(* CoDeSys 2.3.9.62 project: Practica1Ej2.pro *)
(* Libraries: Standard.lib 4.10.05 11:14:46, IecSfc.lib 2.6.14 11:37:46 *)

(* Global variable list: Global_Variables *)
VAR_GLOBAL
     (* Variables de entrada *)
      START:BOOL;
	A:BOOL;
	B:BOOL;
      CC:BOOL;  (*Botón para comienzo de carga*)
      FC:BOOL;   (*Botçon para fin de carga *)
      (* Variables de salida *)
	MOTOR_IZ:BOOL;
	MOTOR_DE:BOOL;
      Carga:BOOL;

       (* Variables para la simulación *)
	Vel:INT:=1;
END_VAR

(* POU PLC_PRG, FBD *)
PROGRAM PLC_PRG
VAR

END_VAR
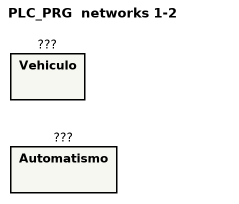
_FBD_ (* Function Block Diagram *)
NETWORK 1
	???:Vehiculo()
NETWORK 2
	???:Automatismo()
_END_FBD_
END_PROGRAM

(* POU Vehiculo, ST *)
PROGRAM Vehiculo
VAR
	PosX: INT;
END_VAR
A:=FALSE;
B:=FALSE;


IF MOTOR_DE=TRUE THEN

     PosX:=PosX+Vel;

END_IF

IF MOTOR_IZ=TRUE THEN

     PosX:=PosX-Vel;

END_IF


IF PosX<=0 THEN
   A:=TRUE;
END_IF

IF PosX>=400 THEN
  B:=TRUE;
END_IF
END_PROGRAM

(* POU Automatismo, LD *)
PROGRAM Automatismo
VAR

END_VAR
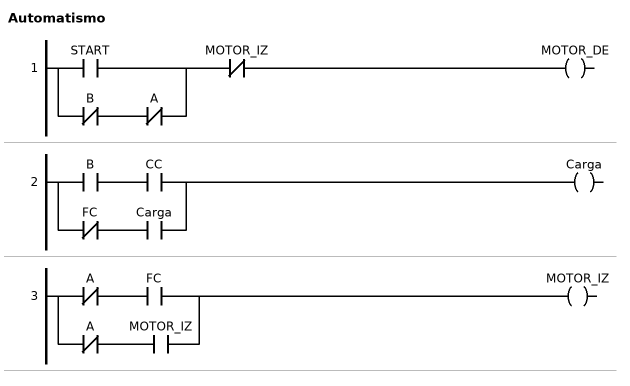
_LD_ (* Ladder Diagram *)
NETWORK 1
	{ [START] | [/B] - [/A] } - [/MOTOR_IZ] --- (MOTOR_DE)
NETWORK 2
	{ [B] - [CC] | [/FC] - [Carga] } --- (Carga)
NETWORK 3
	{ [/A] - [FC] | [/A] - [MOTOR_IZ] } --- (MOTOR_IZ)
_END_LD_
(* the same logic as Structured Text *)
(* Network 1 *)
MOTOR_DE := (START OR NOT B AND NOT A) AND NOT MOTOR_IZ;
(* Network 2 *)
Carga := B AND CC OR NOT FC AND Carga;
(* Network 3 *)
MOTOR_IZ := NOT A AND FC OR NOT A AND MOTOR_IZ;
END_PROGRAM

(* Visualisation Vehiculo
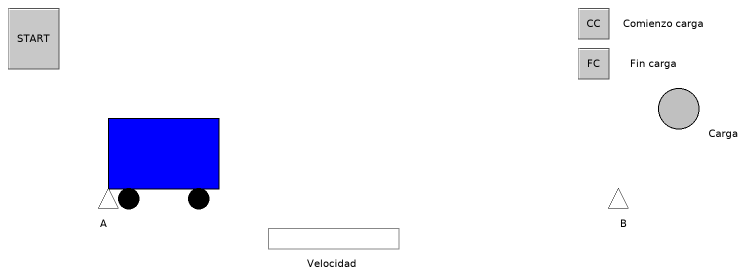
rectangle at (140,120)-(251,191): x offset Vehiculo.PosX
polygon at (130,190)-(150,210): alarm colour if .A
polygon at (640,190)-(660,210): alarm colour if .B
button at (40,10)-(91,71): text "START"; taps START
ellipse at (150,190)-(171,211): x offset Vehiculo.PosX
ellipse at (220,190)-(241,211): x offset Vehiculo.PosX
rectangle at (310,250)-(421,281): text "Velocidad"
rectangle at (80,210)-(191,241): text "A"
rectangle at (600,210)-(711,241): text "B"
button at (610,10)-(641,41): text "CC"; taps CC
button at (610,50)-(641,81): text "FC"; taps FC
ellipse at (690,90)-(731,131): alarm colour if Carga
rectangle at (640,10)-(751,41): text "Comienzo carga"
rectangle at (650,50)-(721,81): text "Fin carga"
rectangle at (700,120)-(811,151): text "Carga"
1 more shapes without text or variables
*)
